// TIA Portal V20 export
DATA_BLOCK "GLOBAL_USER_ALARM_HMI_IF_DB"   // DB219
{ S7_Optimized_Access := 'TRUE' }
// stored: AutoNumber false, MemoryReserve 100
   VAR
      GLOBAL_USER_ALARM : Array[1..30] of "TEC_UNIT_HMI_UDT";
   END_VAR
BEGIN
END_DATA_BLOCK
